// TwinCAT 3 PLC project WinchHyd
// ProgramVersion: 3.1.4023.0
// libraries:
//   Tc2_Standard, * (Beckhoff Automation GmbH)
//   Tc2_System, * (Beckhoff Automation GmbH)
//   Tc3_Module, * (Beckhoff Automation GmbH)
// project tree:
//   CtrlBox/ E_StatusSettings.TcDUT, G_CtrlBoxVariables.TcGVL, ST_BoxParams.TcDUT
//   CtrlBox/FBs + Methods/ FB_BoxSelect.TcPOU, FB_Status.TcPOU
//   CtrlBox/JoyStick/ FB_JoyInputScale.TcPOU, ST_JoyInputScale.TcDUT, ST_ValveScale.TcDUT
//   CtrlBox/MotionControl/ FB_Encoder.TcPOU, ST_WinchCylParams.TcDUT, FB_ValveOutput.TcPOU, FB_WinchControl.TcPOU
//   / GlobalTextList.TcGTLO, PlcTask.TcTTO, Visualization Manager.TcVMO (not stored)
//   Glob_Inputs/ G_Inputs.TcGVL, ST_PressureSensor.TcDUT
//   Glob_Outputs/ G_Outputs.TcGVL
//   HMIControls/ GVL_HMIvars.TcGVL, ST_Enabeling.TcDUT
//   POUs/ MAIN.TcPOU
//   VISUs/Winch/ HMI_winch.TcVIS

CONFIGURATION WinchHyd
    RESOURCE PLC ON TwinCAT3
        TASK PlcTask(INTERVAL := T#10ms, PRIORITY := 20);
        PROGRAM MAIN WITH PlcTask : MAIN;
    END_RESOURCE
END_CONFIGURATION

// ---- CtrlBox/E_StatusSettings.TcDUT
{attribute 'qualified_only'}
{attribute 'strict'}
TYPE E_StatusSettings :
(
	NotReady := 0,
	Ready := 1,
	Starting := 2,
	Running := 3,
	Stopping := 4,
	Fault := 5
);
END_TYPE

// ---- CtrlBox/JoyStick/ST_JoyInputScale.TcDUT
TYPE ST_JoyInputScale :
STRUCT
	fMaxInputVal : REAL := 20509.0;
	fMinInputVal : REAL := 11787.0;
	fNeutralInputVal : REAL := 16175; 
	fNeutralDeadband : REAL := 50.0;
	fMaxOutputValue : REAL := 1.0;
	fMinOutputValue : REAL := -1.0;
	fNeutralOutputValue : REAL := 0.0;
END_STRUCT
END_TYPE

// ---- CtrlBox/JoyStick/ST_ValveScale.TcDUT
TYPE ST_ValveScale :
STRUCT
	fPosMax :LREAL := 29490.0;
	fPosMin : LREAL := 20950.0;
	fNegMin : LREAL := 18250.0;
	fNegMax : LREAL := 9830.0;
END_STRUCT
END_TYPE

// ---- CtrlBox/MotionControl/ST_WinchCylParams.TcDUT
TYPE ST_WinchCylParams :
STRUCT
	fEncoderOffset : UDINT; 
	fDrumDiameter : REAL := 0.475; // m
	fWireDiameter : REAL := 0.014; // m
	fCylStroke : REAL := 0.5; // m
	fRodDiameter : REAL := 0.035; //m
	fPistonDiameter : REAL := 0.065; // m
	fGearRatio : REAL := 1/20; 
END_STRUCT
END_TYPE

// ---- CtrlBox/ST_BoxParams.TcDUT
TYPE ST_BoxParams :
STRUCT
	Start : BOOL;
	Stop : BOOL;
	Off : BOOL;
	Auto : BOOL;
	Manual : BOOL;
	TopSwitch : BOOL;
	JOY_X : INT;
	JOY_Y : INT; 
END_STRUCT
END_TYPE

// ---- Glob_Inputs/ST_PressureSensor.TcDUT
TYPE ST_PressureSensor :
STRUCT
	nSupPressure : INT; 
	nReturnPressure : INT; 
	nCylPistonPressure  : INT; 
	nCylRodPressure : INT; 
	nWinchInPressureA : INT; 
	nWinchInPressureA1 : INT; 
	nWinchOutPressureB : INT;
	nWinchOutPressureB1 : INT; 
	nWinchDrainPressure : INT; 
	nWinchInFlow : INT; 
END_STRUCT
END_TYPE

// ---- HMIControls/ST_Enabeling.TcDUT
TYPE ST_Enabeling :
STRUCT
	bWinchEnable : BOOL := FALSE;
	bCylEnable : BOOL := FALSE; 
	bPosEnable : BOOL := FALSE;
	bVelEnable : BOOL := FALSE;
END_STRUCT
END_TYPE

// ---- CtrlBox/G_CtrlBoxVariables.TcGVL
{attribute 'qualified_only'}
VAR_GLOBAL
	BoxControlVariables : ST_BoxParams; 
END_VAR

// ---- Glob_Inputs/G_Inputs.TcGVL
{attribute 'qualified_only'}
VAR_GLOBAL
	nCylPos : INT; 
	nWinchEncoder : INT; 
	PressureSensorVals : ST_PressureSensor; 
	BoxVariables : ST_BoxParams; 
END_VAR

// ---- Glob_Outputs/G_Outputs.TcGVL
{attribute 'qualified_only'}
VAR_GLOBAL
	fCylValveOut : REAL;
	fWinchValveOut : REAL; 
	bGreenLight : BOOL;
	bRedLight : BOOL; 
	bEnableWinchValve : BOOL;
	bEnableCylValve : BOOL; 	
END_VAR

// ---- HMIControls/GVL_HMIvars.TcGVL
{attribute 'qualified_only'}
VAR_GLOBAL
	stEnable : ST_Enabeling; 
END_VAR

// ---- POUs/MAIN.TcPOU
PROGRAM MAIN
VAR
END_VAR

END_PROGRAM

// ---- CtrlBox/FBs + Methods/FB_BoxSelect.TcPOU
FUNCTION_BLOCK FB_BoxSelect
VAR_INPUT
	bManual : BOOL := ST_BoxParams.Manual;
	bAuto : BOOL := ST_BoxParams.Auto; 
END_VAR
VAR_OUTPUT
	bVirtual : BOOL;
	bReal : BOOL; 
END_VAR
VAR
END_VAR

IF bAuto = TRUE THEN
	bVirtual := TRUE;
ELSIF bManual = TRUE THEN
	bReal := TRUE; 
END_IF

END_FUNCTION_BLOCK

// ---- CtrlBox/FBs + Methods/FB_Status.TcPOU
FUNCTION_BLOCK FB_Status
VAR_INPUT
END_VAR
VAR_OUTPUT
END_VAR
VAR
END_VAR

METHOD FC_GetStatus : INT
VAR_INPUT
	bManualMode : BOOL;
	bAutoMode : BOOL;
	bStartButton : BOOL;
	bStopButton : BOOL; 
	fClock : REAL; 
END_VAR
VAR_OUTPUT
	nSetStatus : INT; 
	bGreenLight : BOOL;
	bRedLight : BOOL; 
END_VAR
IF bManualMode AND bAutoMode = FALSE THEN
	nSetStatus := E_StatusSettings.NotReady;
	
ELSIF bManualMode OR bAutoMode = TRUE THEN
	nSetStatus := E_StatusSettings.Ready;
	
ELSIF bStartButton = TRUE AND NOT (nSetStatus = 4) THEN
	nSetStatus := E_StatusSettings.Starting;

ELSIF (bManualMode AND bStartButton = TRUE) OR (bAutoMode AND bStartButton = TRUE AND fClock > 0) THEN
	bGreenLight := TRUE; 
	nSetStatus := E_StatusSettings.Running;
	
ELSIF (bStopButton = TRUE AND nSetStatus = 4) THEN
	nSetStatus := E_StatusSettings.Stopping;
	bRedLight := TRUE;
	bGreenLight := FALSE; 
	
ELSIF (G_Inputs.PressureSensorVals.nSupPressure < 10 OR G_Inputs.PressureSensorVals.nReturnPressure = 0) THEN
	bRedLight := TRUE;
	bGreenLight := FALSE;
	nSetStatus := E_StatusSettings.Fault; // Change Inputs to converted values when done
	
END_IF
END_METHOD

END_FUNCTION_BLOCK

// ---- CtrlBox/JoyStick/FB_JoyInputScale.TcPOU
FUNCTION_BLOCK FB_JoyInputScale
VAR_INPUT
	nJoyX : INT := G_Inputs.nCylPos;
	bIsManual : BOOL;
	stJoyInputScale : ST_JoyInputScale; 
END_VAR

VAR_OUTPUT
	fJoyX_Norm : LREAL;
END_VAR

VAR
	fRawInput : LREAL;
	fTempInput : LREAL;
	fTempOutput : LREAL;
END_VAR

fRawInput := INT_TO_REAL(nJoyX);

fTempInput := fRawInput - stJoyInputScale.fNeutralInputVal; 

IF fTempInput > stJoyInputScale.fNeutralDeadband THEN
	fTempOutput := fTempInput/(stJoyInputScale.fMaxInputVal - stJoyInputScale.fNeutralInputVal); 

ELSIF fTempInput < -stJoyInputScale.fNeutralDeadband THEN
	fTempOutput := fTempInput/(stJoyInputScale.fNeutralInputVal - stJoyInputScale.fMinInputVal);
	
ELSE
	fTempOutput := 0.0; 
END_IF

IF NOT(bIsManual) THEN
	fJoyX_Norm := 0.0;
ELSE
	fJoyX_Norm := LIMIT(stJoyInputScale.fMinOutputValue, fTempOutput, stJoyInputScale.fMaxOutputValue); 
END_IF

END_FUNCTION_BLOCK

// ---- CtrlBox/MotionControl/FB_Encoder.TcPOU
FUNCTION_BLOCK FB_Encoder
VAR_INPUT
	nRawInput : UDINT; 
	stParam : ST_WinchCylParams; 
END_VAR
VAR_OUTPUT
	fPosition : REAL; 
END_VAR
VAR
	nInput : DINT;
	nTempInputDiff : DINT; 
	nCount : DINT;
	nMaxValue30bit : DINT := 1073741823;
	nThreshold30bit : DINT := nMaxValue30bit/2; 
	fScale16bit : LREAL := 360.0/65535.0;
	fTempPos : LREAL; 
END_VAR
VAR PERSISTENT
	nRounds : DINT;
	nRawLast : DINT; 
END_VAR

nInput := UDINT_TO_DINT(nRawInput);

// ENcoder rounds
IF (nTempInputDiff > nThreshold30bit) THEN
	nRounds := nRounds - 1;
END_IF

IF (nTempInputDiff < -nThreshold30bit) THEN
	nRounds := nRounds + 1; 
END_IF

// Count rounds
nCount := nInput + nRounds*nMaxValue30bit; 

// Pos output
fTempPos := DINT_TO_LREAL(nCount)*fScale16bit - stParam.fEncoderOffset; 

// Convert from winch drum positon to verical position. 
fPosition := FC_DrumToPos(fTempPos, 0); // 0 here should be the registered value for zero position

// Set zero position if load is on ground

METHOD FC_DrumToPos : REAL
VAR_INPUT
	 fCurrentWinchPos : LREAL; 
	 fRegisterdZeroPos : LREAL; 
END_VAR
VAR
	stParams : ST_WinchCylParams; 
END_VAR
VAR_OUTPUT
	fLoadPosition : LREAL; 
END_VAR
fLoadPosition := fRegisterdZeroPos + fCurrentWinchPos*stParams.fDrumDiameter; // If f.eks. 1 round, then output is 1 * drum diameter ergo position is positive 0.475 m from zero
// Need a variable to hold the zero position and add this to the load position.
END_METHOD

END_FUNCTION_BLOCK

// ---- CtrlBox/MotionControl/FB_ValveOutput.TcPOU
FUNCTION_BLOCK FB_ValveOutput
VAR_INPUT
	bIsManual : BOOL;
	bDeadBandCompOn : BOOL;
	stValveScale : ST_ValveScale; 
	fNormalizedInput : LREAL; 
END_VAR
VAR_OUTPUT
	bEnableValve : BOOL;
	nOutput : INT; 
END_VAR
VAR
	nOffset : INT := 19660;
	nMaxValue : INT := 29490;
	nMinValue : INT := 9830;
	nTempOutput : INT; 
END_VAR

IF bDeadBandCompOn THEN
	IF fNormalizedInput > 0.0 THEN
		nTempOutput := LREAL_TO_INT(ABS(fNormalizedInput*(stValveScale.fPosMax - stValveScale.fPosMin) + stValveScale.fPosMin));
	ELSIF fNormalizedInput < 0.0 THEN
		nTempOutput := LREAL_TO_INT(ABS(fNormalizedInput*(stValveScale.fNegMax - stValveScale.fNegMin) - stValveScale.fNegMin)); 
	ELSE
		nTempOutput := nOffset; 
	END_IF
	
ELSE
	IF fNormalizedInput > 0.0 THEN
		nTempOutput := LREAL_TO_INT(ABS(fNormalizedInput*(32767.0 - 19660.0) + 19660)); 
	ELSIF fNormalizedInput < 0.0 THEN
		nTempOutput := LREAL_TO_INT(ABS(fNormalizedInput*(0 - 19660.0) - 19660.0)); 
	ELSE
		nTempOutput := nOffset;
	END_IF
END_IF

IF bIsManual THEN
	nOutput := LIMIT(nMinValue, nTempOutput, nMaxValue);
	bEnableValve := TRUE; 
ELSE
	nOutput := nOffset;
	bEnableValve := FALSE; 
END_IF

END_FUNCTION_BLOCK

// ---- CtrlBox/MotionControl/FB_WinchControl.TcPOU
FUNCTION_BLOCK FB_WinchControl
VAR_INPUT
	bWinch : BOOL := ST_Enabeling.bWinchEnable;
	bPosCtrl : BOOL := ST_Enabeling.bPosEnable;
	bVelCtrl : BOOL := ST_Enabeling.bVelEnable;
END_VAR

VAR_OUTPUT
	fGeneratedPath : REAL;
	fPosCtrlSignal : REAL;
	fVelCtrlSignal : REAL; 
END_VAR
VAR
END_VAR

fGeneratedPath := MotionGenerator()

METHOD MotionGenerator : REAL
VAR_INPUT
	x0: LREAL;
	v_0: LREAL;
	x_ref: LREAL;
	v_ref: LREAL;
	t0: LREAL;
	tRamp: LREAL;
	tWait: LREAL;
	t: LREAL;
END_VAR
VAR_OUTPUT
	x: LREAL;
	v: LREAL;
	Error: LREAL;
END_VAR
VAR
	Error_0: DINT;
	tHold: LREAL;
	x1: LREAL;
	x4: LREAL;
	a_tmp: LREAL;
	a_tmp_tmp: LREAL;
	a_tmp_0: LREAL;
	a_tmp_tmp_0: LREAL;
	a_tmp_tmp_1: LREAL;
	a_tmp_tmp_2: LREAL;
	x1_tmp: LREAL;
	x4_tmp: LREAL;
END_VAR
(* MATLAB Function: '<Root>/Path_signal_gen' *)
(* MATLAB Function 'Path_signal_gen': '<S1>:1' *)
(* '<S1>:1:3' x_SetPoint = x_ref - x0; *)
(* '<S1>:1:4' vs = v_ref; *)
(* '<S1>:1:5' slopeExt = v_0-vs; *)
(* '<S1>:1:6' slopeRetr = -vs-v_0; *)
(* '<S1>:1:8' as = vs/tRamp; *)
(* Find acceleration *)
(* '<S1>:1:9' s_acc = (vs^2-v_0^2)/as; *)
(* Acceleration sp *)
(* '<S1>:1:11' tHold = (x_SetPoint-s_acc)/vs; *)
tHold := ((x_ref - x0) - (((v_ref * v_ref) - (v_0 * v_0)) / (v_ref / tRamp))) / v_ref;
(* '<S1>:1:13' if tHold < 0 *)

IF tHold < 0.0 THEN 
    (* '<S1>:1:14' Error = 1; *)
    Error_0 := 1;
ELSE 
    (* '<S1>:1:15' else *)
    (* '<S1>:1:16' Error = 0; *)
    Error_0 := 0;
END_IF;

(* '<S1>:1:19' t1 = tRamp; *)
(* '<S1>:1:20' t2 = tHold; *)
(* '<S1>:1:21' t3 = tRamp; *)
(* '<S1>:1:22' t4 = tWait; *)
(* '<S1>:1:23' t5 = t1; *)
(* '<S1>:1:24' t6 = t2; *)
(* '<S1>:1:25' t7 = t3; *)
(* Ramp Equations: *)
(* '<S1>:1:28' x1 = x0 + v_0*((t0+t1)-t0) - (slopeExt/t1)*((t0+t1)-t0)^2/2; *)
a_tmp_tmp := t0 + tRamp;
a_tmp := a_tmp_tmp - t0;
x1_tmp := (v_0 - v_ref) / tRamp;
x1 := ((a_tmp * v_0) + x0) - ((x1_tmp * (a_tmp * a_tmp)) / 2.0);
(* '<S1>:1:29' x2 = x1 + vs * ((t0+t1+t2)-(t0+t1)); *)
(* '<S1>:1:30' x4 = x_ref - v_0 * ((t0+t1+t2+t3+t4+t5)-(t0+t1+t2+t3+t4)) + (slopeRetr/t5)*((t0+t1+t2+t3+t4+t5)-(t0+t1+t2+t3+t4))^2/2; *)
a_tmp_tmp_0 := a_tmp_tmp + tHold;
a_tmp_tmp_1 := a_tmp_tmp_0 + tRamp;
a_tmp := a_tmp_tmp_1 + tWait;
a_tmp_tmp_2 := a_tmp + tRamp;
a_tmp_0 := a_tmp_tmp_2 - a_tmp;
x4_tmp := (( -v_ref) - v_0) / tRamp;
x4 := (x_ref - (a_tmp_0 * v_0)) + ((x4_tmp * (a_tmp_0 * a_tmp_0)) / 2.0);
(* '<S1>:1:31' x5 = x4 - vs*((t0+t1+t2+t3+t4+t5+t6)-(t0+t1+t2+t3+t4+t5)); *)
(* '<S1>:1:33' if Error == 1 *)

IF Error_0 = 1 THEN 
    (* Outport: '<Root>/x' *)
    (* '<S1>:1:34' x = x0; *)
    x := x0;
    (* Outport: '<Root>/v' *)
    (* '<S1>:1:35' v = v_0; *)
    v := v_0;
ELSIF (t >= 0.0) AND (t < t0) THEN 
    (* Outport: '<Root>/x' *)
    (* '<S1>:1:36' elseif t >= 0 && t<t0 *)
    (* '<S1>:1:37' x = x0; *)
    x := x0;
    (* Outport: '<Root>/v' *)
    (* '<S1>:1:38' v = v_0; *)
    v := v_0;
ELSIF (t >= t0) AND (t < a_tmp_tmp) THEN 
    (* '<S1>:1:39' elseif t >= t0 && t < (t0+t1) *)
    (* '<S1>:1:40' x = x0 + v_0*(t-t0) - (slopeExt/t1)*(t-t0)^2/2; *)
    a_tmp := t - t0;
    (* Outport: '<Root>/x' *)
    x := ((a_tmp * v_0) + x0) - ((x1_tmp * (a_tmp * a_tmp)) / 2.0);
    (* Outport: '<Root>/v' *)
    (* '<S1>:1:41' v = v_0 - (slopeExt/t1)*(t-t0); *)
    v := v_0 - (x1_tmp * a_tmp);
ELSIF (t >= a_tmp_tmp) AND (t < a_tmp_tmp_0) THEN 
    (* Outport: '<Root>/x' *)
    (* '<S1>:1:42' elseif t >=(t0+t1) && t < (t0+t1+t2) *)
    (* '<S1>:1:43' x = x1 + vs*(t-(t0+t1)); *)
    x := ((t - a_tmp_tmp) * v_ref) + x1;
    (* Outport: '<Root>/v' *)
    (* '<S1>:1:44' v = vs; *)
    v := v_ref;
ELSIF (t >= a_tmp_tmp_0) AND (t < a_tmp_tmp_1) THEN 
    (* '<S1>:1:45' elseif t>=(t0+t1+t2) && t<(t0+t1+t2+t3) *)
    (* '<S1>:1:46' x = x2 + vs*(t-(t0+t1+t2)) + (slopeExt/t3)*(t-(t0+t1+t2))^2/2; *)
    a_tmp := t - a_tmp_tmp_0;
    (* Outport: '<Root>/x' *)
    x := ((((a_tmp_tmp_0 - a_tmp_tmp) * v_ref) + x1) + (a_tmp * v_ref)) + ((x1_tmp * (a_tmp * a_tmp)) / 2.0);
    (* Outport: '<Root>/v' *)
    (* '<S1>:1:47' v = vs + (slopeExt/t3)*(t-(t0+t1+t2)); *)
    v := (a_tmp * x1_tmp) + v_ref;
ELSIF (t >= a_tmp_tmp_1) AND (t < a_tmp) THEN 
    (* Outport: '<Root>/x' *)
    (* '<S1>:1:48' elseif t >=(t0+t1+t2+t3) && t<(t0+t1+t2+t3+t4) *)
    (* '<S1>:1:49' x = x_ref; *)
    x := x_ref;
    (* Outport: '<Root>/v' *)
    (* '<S1>:1:50' v = v_0; *)
    v := v_0;
ELSIF (t >= a_tmp) AND (t < a_tmp_tmp_2) THEN 
    (* '<S1>:1:51' elseif t>=(t0+t1+t2+t3+t4) && t < (t0+t1+t2+t3+t4+t5) *)
    (* '<S1>:1:52' x = x_ref - v_0*(t-(t0+t1+t2+t3+t4))+(slopeRetr/t5)*(t-(t0+t1+t2+t3+t4))^2/2; *)
    a_tmp := t - a_tmp;
    (* Outport: '<Root>/x' *)
    x := (x_ref - (a_tmp * v_0)) + ((x4_tmp * (a_tmp * a_tmp)) / 2.0);
    (* Outport: '<Root>/v' *)
    (* '<S1>:1:53' v = v_0 + (slopeRetr/t5)*(t-(t0+t1+t2+t3+t4)); *)
    v := (a_tmp * x4_tmp) + v_0;
ELSE 
    x1_tmp := a_tmp_tmp_2 + tHold;

    IF (t >= a_tmp_tmp_2) AND (t < x1_tmp) THEN 
        (* Outport: '<Root>/x' *)
        (* '<S1>:1:54' elseif t>=(t0+t1+t2+t3+t4+t5) && t < (t0+t1+t2+t3+t4+t5+t6) *)
        (* '<S1>:1:55' x = x4 - vs*(t-(t0+t1+t2+t3+t4+t5)); *)
        x := x4 - ((t - a_tmp_tmp_2) * v_ref);
        (* Outport: '<Root>/v' *)
        (* '<S1>:1:56' v = -vs; *)
        v :=  -v_ref;
    ELSIF (t >= x1_tmp) AND (t < (x1_tmp + tRamp)) THEN 
        (* '<S1>:1:57' elseif t >= (t0+t1+t2+t3+t4+t5+t6) && t < (t0+t1+t2+t3+t4+t5+t6+t7) *)
        (* '<S1>:1:58' x = x5 - vs*(t-(t0+t1+t2+t3+t4+t5+t6)) - (slopeRetr/t3)*(t-(t0+t1+t2+t3+t4+t5+t6))^2/2; *)
        a_tmp := t - x1_tmp;
        (* Outport: '<Root>/x' *)
        x := ((x4 - ((x1_tmp - a_tmp_tmp_2) * v_ref)) - (a_tmp * v_ref)) - ((x4_tmp * (a_tmp * a_tmp)) / 2.0);
        (* Outport: '<Root>/v' *)
        (* '<S1>:1:59' v = -vs-(slopeRetr/t3)*(t-(t0+t1+t2+t3+t4+t5+t6)); *)
        v := ( -v_ref) - (a_tmp * x4_tmp);
    ELSE 
        (* Outport: '<Root>/x' *)
        (* '<S1>:1:60' else *)
        (* '<S1>:1:61' x = x0; *)
        x := x0;
        (* Outport: '<Root>/v' *)
        (* '<S1>:1:62' v = v_0; *)
        v := v_0;
    END_IF;

END_IF;

(* Outport: '<Root>/Error' incorporates:
 *  MATLAB Function: '<Root>/Path_signal_gen' *)
Error := DINT_TO_LREAL(Error_0);
END_METHOD

METHOD PosControl : REAL
VAR_INPUT
	Enable: LREAL;
	KpGain: LREAL;
	PosRef: LREAL;
	Pos_feedback: LREAL;
END_VAR
VAR_OUTPUT
	Ctrl_signal_Pos: LREAL;
	PosErr: LREAL;
END_VAR
VAR
END_VAR
(* Outputs for Atomic SubSystem: '<Root>/Closed-loop PosCtrl (Auto)' *)
(* Sum: '<S1>/Sum' *)
PosErr := PosRef - Pos_feedback;
(* Product: '<S1>/Product' *)
Ctrl_signal_Pos := KpGain * PosErr;
(* Saturate: '<S1>/Predefined Saturation' *)

IF Ctrl_signal_Pos > 1.0 THEN 
    Ctrl_signal_Pos := 1.0;
ELSIF Ctrl_signal_Pos < -1.0 THEN 
    Ctrl_signal_Pos := -1.0;
END_IF;

(* End of Saturate: '<S1>/Predefined Saturation' *)


(* Switch: '<S1>/Switch' *)

IF Enable <= 0.0 THEN 
    (* Outport: '<Root>/Ctrl_signal_Pos' incorporates:
     *  Constant: '<S1>/Constant' *)
    Ctrl_signal_Pos := 0.0;
END_IF;

(* End of Switch: '<S1>/Switch' *)
(* End of Outputs for SubSystem: '<Root>/Closed-loop PosCtrl (Auto)' *)
END_METHOD

METHOD VelControl : REAL
VAR_INPUT
	vel_refms: LREAL;
	Enable_Signal: LREAL;
	QMax_refLMIN: LREAL;
END_VAR
VAR_OUTPUT
	Ctrl_signalms: LREAL;
END_VAR
VAR
	rtb_Switch: LREAL;
END_VAR
(* Outputs for Atomic SubSystem: '<Root>/Open-loop VelControl (Manual)' *)
(* Switch: '<S1>/Switch' incorporates:
 *  Constant: '<S1>/Annulus_Area'
 *  Constant: '<S1>/Boreside_Area'
 *  Product: '<S1>/Product'
 *  Product: '<S1>/Product1' *)

IF vel_refms > 0.0 THEN 
    rtb_Switch := 0.0033183 * vel_refms;
ELSE 
    rtb_Switch := vel_refms * 0.0023562;
END_IF;

(* End of Switch: '<S1>/Switch' *)


(* Switch: '<S1>/Switch1' incorporates:
 *  Constant: '<S1>/Constant'
 *  Gain: '<S1>/UnitConv'
 *  Product: '<S1>/Divide' *)

IF Enable_Signal > 0.0 THEN 
    Ctrl_signalms := (60000.0 * rtb_Switch) / QMax_refLMIN;
ELSE 
    Ctrl_signalms := 0.0;
END_IF;

(* End of Switch: '<S1>/Switch1' *)


(* Saturate: '<S1>/Saturation' *)

IF Ctrl_signalms > 0.05 THEN 
    (* Outport: '<Root>/Ctrl_signal(m//s)' *)
    Ctrl_signalms := 0.05;
ELSIF Ctrl_signalms < -0.05 THEN 
    (* Outport: '<Root>/Ctrl_signal(m//s)' *)
    Ctrl_signalms := -0.05;
END_IF;

(* End of Saturate: '<S1>/Saturation' *)
(* End of Outputs for SubSystem: '<Root>/Open-loop VelControl (Manual)' *)
END_METHOD

END_FUNCTION_BLOCK

// ---- GlobalTextList.TcGTLO
TEXTLIST GlobalTextList
  268 = 'bEnableWinch'
  709 = 'Enable winch'
  412 = 'Enable Winch'
END_TEXTLIST

// ---- VISUs/Winch/HMI_winch.TcVIS
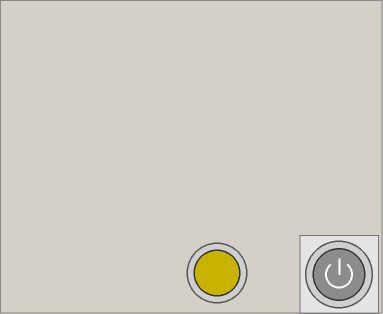
VISUALIZATION HMI_winch  // 383x314
    PowerSwitch (295,235 88x79), variable: GVL_HMIvars.stEnable.bWinchEnable, behaviour: TOGGLE, style: Switch-PowerSwitch-Gray
    Lamp1 (182,238 70x70), variable: GVL_HMIvars.stEnable.bWinchEnable, style: Lamp-Lamp1-Yellow
END_VISUALIZATION
